Universal Robots PolyScope program: regular insertion.urp

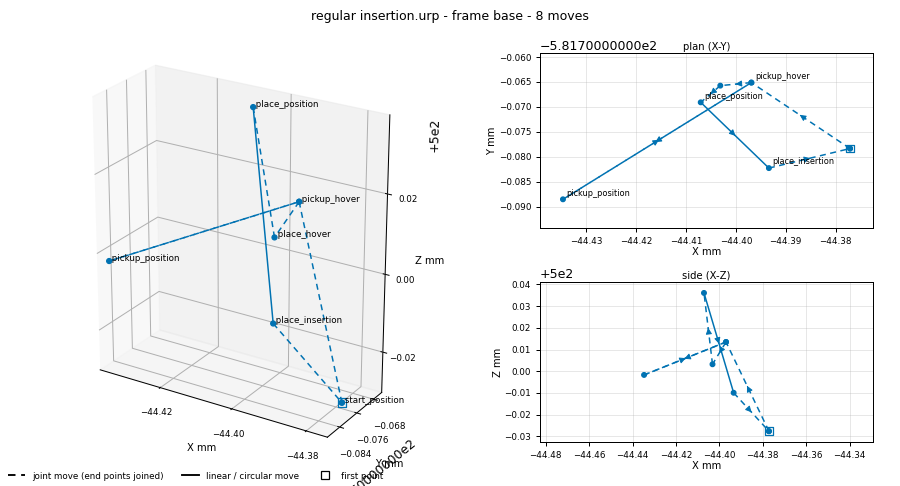
[picture p0: tool path of regular insertion.urp in frame base, 8 of 8 moves have a stored position in this frame; points joined in program order, loops and branches not executed]
Program regular insertion (createdIn=3.2.19293.0 lastSavedIn=3.5.0.10584 directory=/programs installation=default robotSerialNumber=2016352577)
Calibrated DH parameters: a=[0.000176, -0.30042, -0.37922, 0.000042, 0.000063, 0]; d=[0.089415, 194.329143, -181.748083, -12.470753, 0.09493, 0.082587]; alpha=[1.570535, -0.00155, 0.008062, 1.570056, -1.571015, 0]; deltaTheta=[-0.000017, -0.786835, 1.048193, -0.261404, -0.000054, -0.000059]
BeforeStart
  stop_timer := False
  timer := 0
Robot Program (runOnlyOnce=false motionType=MoveJ speed=1.047198 acceleration=1.396263 useActiveTCP=false)
  MoveJ speed 60 deg/s, acceleration 80 deg/s^2 (useActiveTCP=false)
    Waypoint start_position: TCP in base x=-44.377 y=-581.778 z=499.972 mm, rx=-2.2416 ry=-2.1928 rz=-0.0326 rad; joints [74.571, -76.985, 64.998, -76.841, -89.183, 75.97] deg
  URCap Gripper (Robotiq_2-Finger_Adaptive_Gripper, Robotiq Inc.) dataModel(position=0, force=100, speed=100, blocking=true, slaveIds=[9])
  MoveJ speed 60 deg/s, acceleration 80 deg/s^2 (useActiveTCP=false)
    Waypoint pickup_hover: TCP in base x=-44.397 y=-581.765 z=500.013 mm, rx=-2.2417 ry=-2.1928 rz=-0.0324 rad; joints [74.571, -76.985, 64.998, -76.841, -89.183, 75.97] deg; flange x=-44.395 y=-581.808 z=499.976 mm, rx=-2.2418 ry=-2.1927 rz=-0.0324 rad
  URCap Gripper (Robotiq_2-Finger_Adaptive_Gripper, Robotiq Inc.) dataModel(position=68, force=100, speed=100, blocking=true, slaveIds=[9])
  MoveJ speed 60 deg/s, acceleration 80 deg/s^2 (useActiveTCP=false)
    Waypoint pickup_position: TCP in base x=-44.435 y=-581.789 z=499.998 mm, rx=-2.2418 ry=-2.1928 rz=-0.0324 rad; joints [74.571, -76.985, 64.998, -76.841, -89.183, 75.97] deg
  URCap Gripper (Robotiq_2-Finger_Adaptive_Gripper, Robotiq Inc.) dataModel(position=100, force=100, speed=100, blocking=true, slaveIds=[9])
  MoveJ speed 60 deg/s, acceleration 80 deg/s^2 (useActiveTCP=false)
    Waypoint pickup_hover: TCP in base x=-44.397 y=-581.765 z=500.013 mm, rx=-2.2417 ry=-2.1928 rz=-0.0324 rad; joints [74.571, -76.985, 64.998, -76.841, -89.183, 75.97] deg; flange x=-44.395 y=-581.808 z=499.976 mm, rx=-2.2418 ry=-2.1927 rz=-0.0324 rad
  MoveJ speed 60 deg/s, acceleration 80 deg/s^2 (useActiveTCP=false)
    Waypoint place_hover: TCP in base x=-44.403 y=-581.766 z=500.003 mm, rx=-2.2417 ry=-2.1928 rz=-0.0324 rad; joints [74.571, -76.985, 64.998, -76.841, -89.183, 75.97] deg; flange x=-44.395 y=-581.808 z=499.976 mm, rx=-2.2418 ry=-2.1927 rz=-0.0324 rad
  MoveJ speed 60 deg/s, acceleration 80 deg/s^2 (useActiveTCP=false)
    Waypoint place_position: TCP in base x=-44.407 y=-581.769 z=500.036 mm, rx=-2.2417 ry=-2.1928 rz=-0.0322 rad; joints [74.571, -76.985, 64.998, -76.841, -89.183, 75.97] deg; flange x=-44.395 y=-581.808 z=499.976 mm, rx=-2.2418 ry=-2.1927 rz=-0.0324 rad
  MoveL speed 250 mm/s, acceleration 1200 mm/s^2 (useActiveTCP=false) feature=Base
    Waypoint place_insertion: TCP in base x=-44.393 y=-581.782 z=499.99 mm, rx=-2.2417 ry=-2.1928 rz=-0.0324 rad; joints [74.571, -76.985, 64.998, -76.841, -89.183, 75.97] deg
  URCap Gripper (Robotiq_2-Finger_Adaptive_Gripper, Robotiq Inc.) dataModel(position=0, force=100, speed=100, blocking=true, slaveIds=[9])
  MoveJ speed 60 deg/s, acceleration 80 deg/s^2 (useActiveTCP=false)
    Waypoint start_position: TCP in base x=-44.377 y=-581.778 z=499.972 mm, rx=-2.2416 ry=-2.1928 rz=-0.0326 rad; joints [74.571, -76.985, 64.998, -76.841, -89.183, 75.97] deg
  Halt
Thread Thread_1 (runOnlyOnce=false trackProgramExecution=false)
  sensor_data := socket_read_ascii_float(6,"stream")
  If sensor_data[0] ≥6
    Fx := sensor_data[1]   [initializeExpression=0.0]
    Fy := sensor_data[2]   [initializeExpression=0.0]
    Fz := sensor_data[3]   [initializeExpression=0.0]
    Mx := sensor_data[4]   [initializeExpression=0.0]
    My := sensor_data[5]   [initializeExpression=0.0]
    Mz := sensor_data[6]   [initializeExpression=0.0]
  Else 
    Fx := 0.0
    Fy := 0.0
    Fz := 0.0
    Mx := 0.0
    My := 0.0
    Mz := 0.0
Thread Thread_2 (runOnlyOnce=false trackProgramExecution=false)
  If stop_timer ≟ True
    Script: timer = timer +.008
  Else 
    Script: timer =0
  Wait Sleep waitTime=0.008
